// LS Electric XG5000 project: DAY08
// PLC LSPLC
// module base 0 slot 0: 입출력 모듈:XBC-DR30S (DC 24V 입력 18점, 릴레이 출력 12점)

PROGRAM NewProgram (task: 스캔 프로그램)

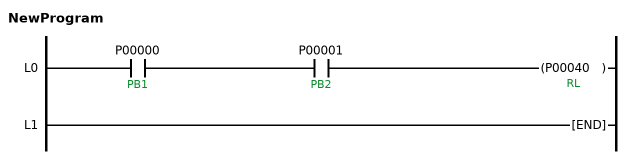
; L0
LOAD      P00000	// PB1
AND       P00001	// PB2
OUT       P00040	// RL
; L1
END